// TIA Portal V15.1 export
// export: Created 2026-01-15T16:29:48.9284817Z, ExportSetting WithDefaults, WithReadOnly, DisplayName Totally Integrated Automation Portal, DisplayVersion V15.1 Update 8, DisplayName TIA Portal Openness, DisplayVersion V15.1 Update 8, DisplayName STEP 7 Professional, DisplayVersion V15.1 Update 8, DisplayName WinCC Advanced, DisplayVersion V15.1 Update 8
VAR_GLOBAL   // PLC tag table "XUNG_TEMP"
   P_AGG1_EM AT %M100.0 : Bool;
   P_AGG2_EM AT %M100.1 : Bool;
   P_AGG3_EM AT %M100.2 : Bool;
   P_AGG4_EM AT %M100.3 : Bool;
   P_AGG5_EM AT %M100.4 : Bool;
   P_AGG6_EM AT %M100.5 : Bool;
   P_CE1_EM AT %M100.6 : Bool;
   P_CE2_EM AT %M100.7 : Bool;
   P_CE3_EM AT %M101.0 : Bool;
   P_CE4_EM AT %M101.1 : Bool;
   P_CE5_EM AT %M101.2 : Bool;
   P_WA1_EM AT %M101.3 : Bool;
   P_WA2_EM AT %M101.4 : Bool;
   P_ADD1_EM AT %M101.5 : Bool;
   P_ADD2_EM AT %M101.6 : Bool;
   P_ADD3_EM AT %M101.7 : Bool;
   P_ADD4_EM AT %M102.0 : Bool;
   P_ADD5_EM AT %M102.1 : Bool;
   P_ADD6_EM AT %M102.2 : Bool;
   P_WAGG1_EM AT %M102.3 : Bool;
   P_WAGG2_EM AT %M102.4 : Bool;
   P_WAGG3_EM AT %M102.5 : Bool;
   P_WAGG4_EM AT %M102.6 : Bool;
   P_WAGG5_EM AT %M102.7 : Bool;
   P_WAGG6_EM AT %M103.0 : Bool;
   P_WCEM1_EM AT %M103.1 : Bool;
   P_WCEM2_EM AT %M103.2 : Bool;
   P_WWAT1_EM AT %M103.3 : Bool;
   P_WWAT2_EM AT %M103.4 : Bool;
   P_WADD1_EM AT %M103.5 : Bool;
   P_WADD2_EM AT %M103.6 : Bool;
   P_AGG1_FU AT %M103.7 : Bool;
   P_AGG2_FU AT %M104.0 : Bool;
   P_AGG3_FU AT %M104.1 : Bool;
   P_AGG4_FU AT %M104.2 : Bool;
   P_AGG5_FU AT %M104.3 : Bool;
   P_AGG6_FU AT %M104.4 : Bool;
   P_CE1_FU AT %M104.5 : Bool;
   P_CE2_FU AT %M104.6 : Bool;
   P_CE3_FU AT %M104.7 : Bool;
   P_CE4_FU AT %M105.0 : Bool;
   P_CE5_FU AT %M105.1 : Bool;
   P_WA1_FU AT %M105.2 : Bool;
   P_WA2_FU AT %M105.3 : Bool;
   P_ADD1_FU AT %M105.4 : Bool;
   P_ADD2_FU AT %M105.5 : Bool;
   P_ADD3_FU AT %M105.6 : Bool;
   P_ADD4_FU AT %M105.7 : Bool;
   P_ADD5_FU AT %M106.0 : Bool;
   P_ADD6_FU AT %M106.1 : Bool;
   P_WAGG1_FU AT %M106.2 : Bool;
   P_WAGG2_FU AT %M106.3 : Bool;
   P_WAGG3_FU AT %M106.4 : Bool;
   P_WAGG4_FU AT %M106.5 : Bool;
   P_WAGG5_FU AT %M106.6 : Bool;
   P_WAGG6_FU AT %M106.7 : Bool;
   P_WCEM1_FU AT %M107.0 : Bool;
   P_WCEM2_FU AT %M107.1 : Bool;
   P_WWAT1_FU AT %M107.2 : Bool;
   P_WWAT2_FU AT %M107.3 : Bool;
   P_WADD1_FU AT %M107.4 : Bool;
   P_WADD2_FU AT %M107.5 : Bool;
   P_PTG_EM AT %M107.6 : Bool;
   P_PTG_FU AT %M107.7 : Bool;
   P_SKIP_EM AT %M108.0 : Bool;
   P_SKIP_FU AT %M108.1 : Bool;
   P_MIXER_EM AT %M108.2 : Bool;
   P_MIXER_FU AT %M108.3 : Bool;
   P_RUN AT %M108.4 : Bool;
   "P_COT LIEU_FU" AT %M108.5 : Bool;
   "P_COT LIEU_EM" AT %M108.6 : Bool;
   "P_XA AGG1" AT %M108.7 : Bool;
   "P_XA AGG2" AT %M109.0 : Bool;
   "P_XA AGG3" AT %M109.1 : Bool;
   "P_XA AGG4" AT %M109.2 : Bool;
   "P_XA AGG5" AT %M109.3 : Bool;
   "P_XA AGG6" AT %M109.4 : Bool;
   "P_XA PTG" AT %M109.5 : Bool;
   "P_XA CEM1" AT %M109.6 : Bool;
   "P_XA CEM2" AT %M109.7 : Bool;
   "P_XA WAT1" AT %M110.0 : Bool;
   "P_XA WAT2" AT %M110.1 : Bool;
   "P_XA ADD1" AT %M110.2 : Bool;
   "P_XA ADD2" AT %M110.3 : Bool;
END_VAR
